VAR_GLOBAL

	fbAct1:FB_ActionneurSimple;	//Act1 corresponds to charging
	fbAct2:FB_ActionneurSimple;	//Act2 corresponds to engraving
	fbAct3:FB_ActionneurSimple;	//Act3 corresponds to tightening
	
	xModeStepForStep :BOOL;
	xNextStep : BOOL;
	
	//pour FB_gestion du mode
	fbMMA:FB_MMA;
	fbCycleAuto:FB_CycleAuto;
	fbCycleInit : FB_CycleInit;
	fbCycleMan : FB_CycleMan;
	
	stParam:ST_Param;
	fbBtn:FB_Btn;
	stIO:ST_IO;
	
	//Tachymetre moteur
	fbMotor : FB_RegulMoteur;
	
	//include TCP_LIB
	fbTCP : FB_TCP;
	
	//
	fbErrorAdmin:FB_ErrorAdmin;//gestion des erreurs, messages
	fbErrorViewer:FB_ErrorViewer;//gestion de l'affichage du tableau
	

	 
END_VAR

(* stored: Version 1.1.0.1, ProductVersion 3.1.4020.6
   GVL GVL: Id {29e74ae1-1e66-43a7-ba4b-1961dad16adc} *)
